ABB RAPID module: CodigoRAPID

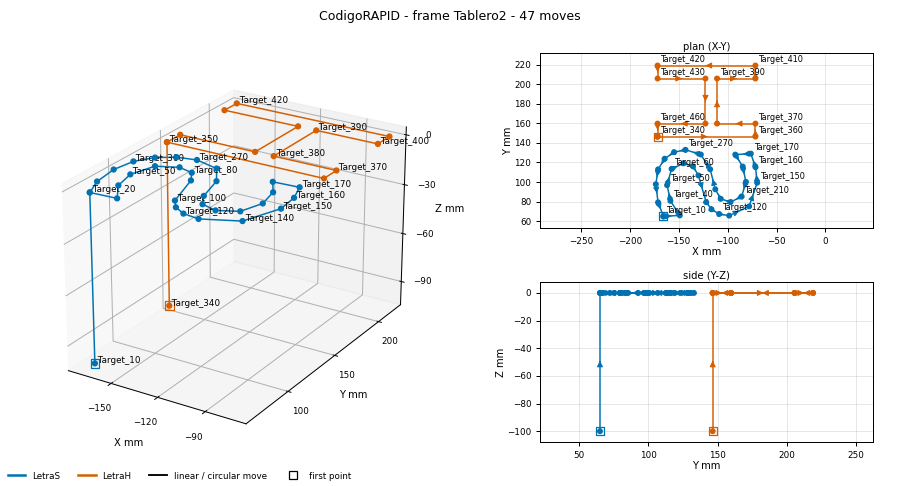
[picture p0: tool path of CodigoRAPID in frame Tablero2, 47 of 50 moves have a stored position in this frame; points joined in program order, loops and branches not executed]
MODULE Module1
        CONST robtarget Target_10:=[[-165.598593277,64.965962784,-99.999795856],[0.332652119,0.000000622,-0.00000022,-0.94304961],[0,0,0,0],[9E+09,9E+09,9E+09,9E+09,9E+09,9E+09]];
    CONST robtarget Target_20:=[[-165.598725349,64.965962784,0.000204144],[0.332652119,0.000000622,-0.00000022,-0.94304961],[0,0,0,0],[9E+09,9E+09,9E+09,9E+09,9E+09,9E+09]];
    CONST robtarget Target_30:=[[-148.905046256,65.938410109,0.000226192],[0.332652119,0.000000623,-0.00000022,-0.94304961],[0,0,0,0],[9E+09,9E+09,9E+09,9E+09,9E+09,9E+09]];
    CONST robtarget Target_40:=[[-158.46744496,80.808750466,0.000213562],[0.332652119,0.000000623,-0.000000219,-0.94304961],[0,0,0,0],[9E+09,9E+09,9E+09,9E+09,9E+09,9E+09]];
    CONST robtarget Target_50:=[[-161.8710106,96.813612703,0.000209067],[0.332652119,0.000000623,-0.00000022,-0.94304961],[0,0,0,0],[9E+09,9E+09,9E+09,9E+09,9E+09,9E+09]];
    CONST robtarget Target_60:=[[-157.292404442,113.466773156,0.000215114],[0.332652119,0.000000622,-0.000000219,-0.94304961],[0,0,0,0],[9E+09,9E+09,9E+09,9E+09,9E+09,9E+09]];
    CONST robtarget Target_70:=[[-145.177331508,119.098863918,0.000231115],[0.332652119,0.000000622,-0.00000022,-0.94304961],[0,0,0,0],[9E+09,9E+09,9E+09,9E+09,9E+09,9E+09]];
    CONST robtarget Target_80:=[[-135.45285825,116.141003302,0.000243958],[0.332652119,0.000000623,-0.000000219,-0.943049611],[0,0,0,0],[9E+09,9E+09,9E+09,9E+09,9E+09,9E+09]];
    CONST robtarget Target_90:=[[-129.861286127,106.781197792,0.000251344],[0.332652119,0.000000622,-0.00000022,-0.94304961],[0,0,0,0],[9E+09,9E+09,9E+09,9E+09,9E+09,9E+09]];
    CONST robtarget Target_100:=[[-121.879114328,79.431116754,0.000261886],[0.332652119,0.000000622,-0.000000219,-0.94304961],[0,0,0,0],[9E+09,9E+09,9E+09,9E+09,9E+09,9E+09]];
    CONST robtarget Target_110:=[[-116.490135398,72.17828045,0.000269002],[0.332652119,0.000000623,-0.00000022,-0.94304961],[0,0,0,0],[9E+09,9E+09,9E+09,9E+09,9E+09,9E+09]];
    CONST robtarget Target_120:=[[-108.710556792,67.397081098,0.000279277],[0.332652119,0.000000623,-0.000000219,-0.94304961],[0,0,0,0],[9E+09,9E+09,9E+09,9E+09,9E+09,9E+09]];
    CONST robtarget Target_130:=[[-98.418822594,65.695298278,0.00029287],[0.332652119,0.000000622,-0.00000022,-0.94304961],[0,0,0,0],[9E+09,9E+09,9E+09,9E+09,9E+09,9E+09]];
    CONST robtarget Target_140:=[[-78.037947391,75.176659704,0.000319788],[0.332652119,0.000000623,-0.00000022,-0.94304961],[0,0,0,0],[9E+09,9E+09,9E+09,9E+09,9E+09,9E+09]];
    CONST robtarget Target_150:=[[-69.812663761,99.325768294,0.000330651],[0.332652119,0.000000623,-0.00000022,-0.94304961],[0,0,0,0],[9E+09,9E+09,9E+09,9E+09,9E+09,9E+09]];
    CONST robtarget Target_160:=[[-71.473927942,115.209074615,0.000328457],[0.33265212,0.000000623,-0.00000022,-0.94304961],[0,0,0,0],[9E+09,9E+09,9E+09,9E+09,9E+09,9E+09]];
    CONST robtarget Target_170:=[[-76.295645932,129.066449007,0.000322089],[0.332652119,0.000000623,-0.00000022,-0.94304961],[0,0,0,0],[9E+09,9E+09,9E+09,9E+09,9E+09,9E+09]];
    CONST robtarget Target_180:=[[-92.178952253,128.094001681,0.000301111],[0.332652119,0.000000623,-0.00000022,-0.94304961],[0,0,0,0],[9E+09,9E+09,9E+09,9E+09,9E+09,9E+09]];
    CONST robtarget Target_190:=[[-84.561448202,115.857372832,0.000311172],[0.332652119,0.000000623,-0.00000022,-0.94304961],[0,0,0,0],[9E+09,9E+09,9E+09,9E+09,9E+09,9E+09]];
    CONST robtarget Target_200:=[[-81.319957116,100.217178343,0.000315453],[0.332652119,0.000000623,-0.00000022,-0.94304961],[0,0,0,0],[9E+09,9E+09,9E+09,9E+09,9E+09,9E+09]];
    CONST robtarget Target_210:=[[-85.655451443,85.265800709,0.000309727],[0.33265212,0.000000622,-0.00000022,-0.94304961],[0,0,0,0],[9E+09,9E+09,9E+09,9E+09,9E+09,9E+09]];
    CONST robtarget Target_220:=[[-97.041188883,79.55267267,0.00029469],[0.332652119,0.000000622,-0.00000022,-0.94304961],[0,0,0,0],[9E+09,9E+09,9E+09,9E+09,9E+09,9E+09]];
    CONST robtarget Target_230:=[[-107.130329887,82.915719672,0.000281365],[0.332652119,0.000000623,-0.00000022,-0.94304961],[0,0,0,0],[9E+09,9E+09,9E+09,9E+09,9E+09,9E+09]];
    CONST robtarget Target_240:=[[-112.600346095,92.599674291,0.000274141],[0.332652119,0.000000622,-0.00000022,-0.94304961],[0,0,0,0],[9E+09,9E+09,9E+09,9E+09,9E+09,9E+09]];
    CONST robtarget Target_250:=[[-117.867769109,113.102105409,0.000267183],[0.33265212,0.000000623,-0.00000022,-0.94304961],[0,0,0,0],[9E+09,9E+09,9E+09,9E+09,9E+09,9E+09]];
    CONST robtarget Target_260:=[[-127.389649174,128.175038959,0.000254608],[0.33265212,0.000000623,-0.00000022,-0.94304961],[0,0,0,0],[9E+09,9E+09,9E+09,9E+09,9E+09,9E+09]];
    CONST robtarget Target_270:=[[-143.070362302,132.95623831,0.000233897],[0.332652119,0.000000622,-0.00000022,-0.94304961],[0,0,0,0],[9E+09,9E+09,9E+09,9E+09,9E+09,9E+09]];
    CONST robtarget Target_280:=[[-154.658692934,130.565638634,0.000218593],[0.33265212,0.000000623,-0.00000022,-0.94304961],[0,0,0,0],[9E+09,9E+09,9E+09,9E+09,9E+09,9E+09]];
    CONST robtarget Target_290:=[[-164.302128915,123.88006327,0.000205856],[0.332652119,0.000000623,-0.000000219,-0.94304961],[0,0,0,0],[9E+09,9E+09,9E+09,9E+09,9E+09,9E+09]];
    CONST robtarget Target_300:=[[-171.028222918,113.021068132,0.000196973],[0.332652119,0.000000622,-0.000000219,-0.94304961],[0,0,0,0],[9E+09,9E+09,9E+09,9E+09,9E+09,9E+09]];
    CONST robtarget Target_310:=[[-173.378303955,97.786060028,0.000193869],[0.332652119,0.000000623,-0.00000022,-0.94304961],[0,0,0,0],[9E+09,9E+09,9E+09,9E+09,9E+09,9E+09]];
    CONST robtarget Target_320:=[[-171.109260196,79.309560839,0.000196866],[0.332652119,0.000000623,-0.000000219,-0.94304961],[0,0,0,0],[9E+09,9E+09,9E+09,9E+09,9E+09,9E+09]];
    CONST robtarget Target_330:=[[-165.598725349,64.965962784,0.000204144],[0.332652119,0.000000622,-0.00000022,-0.94304961],[0,0,0,0],[9E+09,9E+09,9E+09,9E+09,9E+09,9E+09]];
    CONST robtarget Target_340:=[[-171.595351785,146.489463594,-99.999803776],[0.332652097,0.000000622,-0.00000022,-0.943049618],[0,0,0,0],[9E+09,9E+09,9E+09,9E+09,9E+09,9E+09]];
    CONST robtarget Target_350:=[[-171.595483858,146.489463594,0.000196224],[0.332652097,0.000000622,-0.00000022,-0.943049618],[0,0,0,0],[9E+09,9E+09,9E+09,9E+09,9E+09,9E+09]];
    CONST robtarget Target_360:=[[-71.595483858,146.489463594,0.000328296],[0.332652097,0.000000622,-0.00000022,-0.943049618],[0,0,0,0],[9E+09,9E+09,9E+09,9E+09,9E+09,9E+09]];
    CONST robtarget Target_370:=[[-71.595483858,159.779577046,0.000328296],[0.332652097,0.000000623,-0.00000022,-0.943049618],[0,0,0,0],[9E+09,9E+09,9E+09,9E+09,9E+09,9E+09]];
    CONST robtarget Target_380:=[[-110.817525998,159.779577046,0.000276495],[0.332652097,0.000000622,-0.00000022,-0.943049618],[0,0,0,0],[9E+09,9E+09,9E+09,9E+09,9E+09,9E+09]];
    CONST robtarget Target_390:=[[-110.817525998,205.808750466,0.000276495],[0.332652097,0.000000623,-0.00000022,-0.943049618],[0,0,0,0],[9E+09,9E+09,9E+09,9E+09,9E+09,9E+09]];
    CONST robtarget Target_400:=[[-71.595483858,205.808750466,0.000328296],[0.332652097,0.000000622,-0.00000022,-0.943049618],[0,0,0,0],[9E+09,9E+09,9E+09,9E+09,9E+09,9E+09]];
    CONST robtarget Target_410:=[[-71.595483858,219.098863918,0.000328296],[0.332652097,0.000000623,-0.00000022,-0.943049618],[0,0,0,0],[9E+09,9E+09,9E+09,9E+09,9E+09,9E+09]];
    CONST robtarget Target_420:=[[-171.595483858,219.098863918,0.000196224],[0.332652097,0.000000622,-0.00000022,-0.943049618],[0,0,0,0],[9E+09,9E+09,9E+09,9E+09,9E+09,9E+09]];
    CONST robtarget Target_430:=[[-171.595483858,205.808750466,0.000196224],[0.332652097,0.000000623,-0.00000022,-0.943049618],[0,0,0,0],[9E+09,9E+09,9E+09,9E+09,9E+09,9E+09]];
    CONST robtarget Target_440:=[[-122.648968461,205.808750466,0.000260869],[0.332652097,0.000000622,-0.00000022,-0.943049618],[0,0,0,0],[9E+09,9E+09,9E+09,9E+09,9E+09,9E+09]];
    CONST robtarget Target_450:=[[-122.648968461,159.779577046,0.000260869],[0.332652097,0.000000623,-0.00000022,-0.943049618],[0,0,0,0],[9E+09,9E+09,9E+09,9E+09,9E+09,9E+09]];
    CONST robtarget Target_460:=[[-171.595483858,159.779577046,0.000196224],[0.332652097,0.000000622,-0.00000022,-0.943049618],[0,0,0,0],[9E+09,9E+09,9E+09,9E+09,9E+09,9E+09]];
    CONST robtarget Target_470:=[[-171.595483858,146.489463594,0.000196224],[0.332652097,0.000000623,-0.00000022,-0.943049618],[0,0,0,0],[9E+09,9E+09,9E+09,9E+09,9E+09,9E+09]];
    CONST jointtarget Home:=[[0,0,0,0,0,0],[9E+09,9E+09,9E+09,9E+09,9E+09,9E+09]];
    CONST jointtarget Intermedio:=[[0,9.2,20,27.2,33.4,0],[9E+09,9E+09,9E+09,9E+09,9E+09,9E+09]];
    CONST jointtarget CambioHerramienta:=[[90,0,0,0,0,0],[9E+09,9E+09,9E+09,9E+09,9E+09,9E+09]];
!*********************
    !
    ! Módulo:  Module1
    !
    ! Descripción:
    !   <Introduzca la descripción aquí>
    !
    ! Autor: alejo
    !
    ! Versión: 1.0
    !
    !*********************


    !*********************
    !
    ! Procedimiento Main
    !
    !   Este es el punto de entrada de su programa
    !
    !*********************
    PROC main()
        GoHome;
        SetDO Sal1,0;
        WaitDI Ent2,1;
        GoCambio;
        WaitDI Ent1,1;
        GoHome;
        SetDO Sal1,1;
        GoIntermedio;
        LetraS;
        LetraH;
        GoIntermedio;
        GoHome;
    ENDPROC
    PROC LetraS()
        MoveL Target_10,v150,z10,Portamarcador2\WObj:=Tablero2;
        MoveL Target_20,v150,z10,Portamarcador2\WObj:=Tablero2;
        MoveL Target_30,v150,z10,Portamarcador2\WObj:=Tablero2;
        MoveL Target_40,v150,z10,Portamarcador2\WObj:=Tablero2;
        MoveL Target_50,v150,z10,Portamarcador2\WObj:=Tablero2;
        MoveL Target_60,v150,z10,Portamarcador2\WObj:=Tablero2;
        MoveL Target_70,v150,z10,Portamarcador2\WObj:=Tablero2;
        MoveL Target_80,v150,z10,Portamarcador2\WObj:=Tablero2;
        MoveL Target_90,v150,z10,Portamarcador2\WObj:=Tablero2;
        MoveL Target_100,v150,z10,Portamarcador2\WObj:=Tablero2;
        MoveL Target_110,v150,z10,Portamarcador2\WObj:=Tablero2;
        MoveL Target_120,v150,z10,Portamarcador2\WObj:=Tablero2;
        MoveL Target_130,v150,z10,Portamarcador2\WObj:=Tablero2;
        MoveL Target_140,v150,z10,Portamarcador2\WObj:=Tablero2;
        MoveL Target_150,v150,z10,Portamarcador2\WObj:=Tablero2;
        MoveL Target_160,v150,z10,Portamarcador2\WObj:=Tablero2;
        MoveL Target_170,v150,z10,Portamarcador2\WObj:=Tablero2;
        MoveL Target_180,v150,z10,Portamarcador2\WObj:=Tablero2;
        MoveL Target_190,v150,z10,Portamarcador2\WObj:=Tablero2;
        MoveL Target_200,v150,z10,Portamarcador2\WObj:=Tablero2;
        MoveL Target_210,v150,z10,Portamarcador2\WObj:=Tablero2;
        MoveL Target_220,v150,z10,Portamarcador2\WObj:=Tablero2;
        MoveL Target_230,v150,z10,Portamarcador2\WObj:=Tablero2;
        MoveL Target_240,v150,z10,Portamarcador2\WObj:=Tablero2;
        MoveL Target_250,v150,z10,Portamarcador2\WObj:=Tablero2;
        MoveL Target_260,v150,z10,Portamarcador2\WObj:=Tablero2;
        MoveL Target_270,v150,z10,Portamarcador2\WObj:=Tablero2;
        MoveL Target_280,v150,z10,Portamarcador2\WObj:=Tablero2;
        MoveL Target_290,v150,z10,Portamarcador2\WObj:=Tablero2;
        MoveL Target_300,v150,z10,Portamarcador2\WObj:=Tablero2;
        MoveL Target_310,v150,z10,Portamarcador2\WObj:=Tablero2;
        MoveL Target_320,v150,z10,Portamarcador2\WObj:=Tablero2;
        MoveL Target_330,v150,z10,Portamarcador2\WObj:=Tablero2;
    ENDPROC
    PROC LetraH()
        MoveL Target_340,v200,z10,Portamarcador2\WObj:=Tablero2;
        MoveL Target_350,v200,z10,Portamarcador2\WObj:=Tablero2;
        MoveL Target_360,v200,z10,Portamarcador2\WObj:=Tablero2;
        MoveL Target_370,v200,z10,Portamarcador2\WObj:=Tablero2;
        MoveL Target_380,v200,z10,Portamarcador2\WObj:=Tablero2;
        MoveL Target_390,v200,z10,Portamarcador2\WObj:=Tablero2;
        MoveL Target_400,v200,z10,Portamarcador2\WObj:=Tablero2;
        MoveL Target_410,v200,z10,Portamarcador2\WObj:=Tablero2;
        MoveL Target_420,v200,z10,Portamarcador2\WObj:=Tablero2;
        MoveL Target_430,v200,z10,Portamarcador2\WObj:=Tablero2;
        MoveL Target_440,v200,z10,Portamarcador2\WObj:=Tablero2;
        MoveL Target_450,v200,z10,Portamarcador2\WObj:=Tablero2;
        MoveL Target_460,v200,z10,Portamarcador2\WObj:=Tablero2;
        MoveL Target_470,v200,z10,Portamarcador2\WObj:=Tablero2;
    ENDPROC
    PROC GoHome()
        MoveAbsJ Home,v200,z100,Portamarcador2\WObj:=Tablero2;
    ENDPROC
    PROC GoIntermedio()
        MoveAbsJ Intermedio,v200,z100,Portamarcador2\WObj:=Tablero2;
    ENDPROC
    PROC GoCambio()
        MoveAbsJ CambioHerramienta,v200,z100,Portamarcador2\WObj:=Tablero2;
    ENDPROC
ENDMODULE
